// TIA Portal V20 export
// export: Created 2026-04-18T06:33:56.4974019Z, ExportSetting WithDefaults, DisplayName Totally Integrated Automation Portal, DisplayVersion V20, DisplayName TIA Portal Openness, DisplayVersion V20, DisplayName TIA Portal Version Control Interface, DisplayVersion V20, DisplayName STEP 7 Professional, DisplayVersion V20, DisplayName STEP 7 Safety, DisplayVersion V20, DisplayName WinCC Basic/Comfort/Advanced, DisplayVersion V20
TYPE "driveMessagesConfig_UDT"
// stored: IsFailsafeCompliant false
   STRUCT
      communicationError { ExternalAccessible := 'False'; ExternalVisible := 'False'; ExternalWritable := 'False'; S7_SetPoint := 'True'} : "messageConfig_UDT";
      blocked { ExternalAccessible := 'False'; ExternalVisible := 'False'; ExternalWritable := 'False'; S7_SetPoint := 'True'} : "messageConfig_UDT";
   END_STRUCT;
END_TYPE
